{attribute 'linkalways'} 
{attribute 'no_explicit_call' := 'This FB is a CLASS and must be accessed using methods or properties'}
{attribute 'enable_dynamic_creation'}
FUNCTION_BLOCK FINAL AND_UDINT EXTENDS Node
VAR
	in1 : _UDINT(0);
	in2 : _UDINT(0);
	out : _UDINT(0);
END_VAR

METHOD PUBLIC Clone : I_Node
VAR
	pNode : POINTER TO AND_UDINT;
END_VAR
pNode := __NEW(AND_UDINT);
Clone := pNode^;
END_METHOD

METHOD FB_init : BOOL
VAR_INPUT
	bInitRetains : BOOL; // if TRUE, the retain variables are initialized (warm start / cold start)
	bInCopyCode : BOOL;  // if TRUE, the instance afterwards gets moved into the copy code (online change)
END_VAR
AddInput('in1',THIS^.in1);
AddInput('in2',THIS^.in2);
AddOutput('out', THIS^.out);
END_METHOD

METHOD PROTECTED OnExecute
VAR
END_VAR
out.Value := in1.Value AND in2.Value;
END_METHOD

END_FUNCTION_BLOCK

(* stored: Version 1.1.0.1, ProductVersion 3.1.4024.15
   POU AND_UDINT: Id {75321ed8-aa78-4285-b319-3ad7f3b29ace}, SpecialFunc None
   Folder Constructor: Id {b664e72f-d915-409f-96fe-36d0f266fefc}
   Method Clone: Id {a2ab27fb-021a-4bec-8064-898006704e74}
   Method FB_init: Id {ff577cab-18ac-4204-a0c8-7fedea377d32}
   Method OnExecute: Id {da0241fb-86fc-47e5-87cc-fad6d73ffc32} *)
